FUNCTION_BLOCK TTest_LicenceCheck EXTENDS TcUnit.FB_TestSuite
VAR_INPUT
END_VAR
VAR_OUTPUT
END_VAR
VAR
END_VAR

LicenceCheck_GetsValidLicence();
LicenceCheck_GetsInValidLicence();

METHOD LicenceCheck_GetsInValidLicence
VAR_INST
    LicenceCheck : TLicenceCheck(
        LicenceIdAsString      := '{13ae39d9-bbb2-423e-8ace-d2c791a6b0ec}', // 1st digit should be 0
        LicenceName            := 'tcl_BaseLib',
        StopTwinCAT_IfNotValid := FALSE);
END_VAR
TEST(TestName := 'LicenceCheck_GetsInValidLicence');

LicenceCheck();

IF LicenceCheck.CheckComplete THEN
    AssertEquals_BOOL(
        Expected := FALSE,
        Actual   := LicenceCheck.IsValid,
        Message  := 'Licence check failed');
        
    TEST_FINISHED();
END_IF
END_METHOD

METHOD LicenceCheck_GetsValidLicence
VAR_INST
    LicenceCheck : TLicenceCheck(
        LicenceIdAsString      := '{4c256767-e6e6-4af5-bd68-9f7abad0c200}', // Tc_Ads Id
        LicenceName            := 'tcl_BaseLib',
        StopTwinCAT_IfNotValid := FALSE);
END_VAR
TEST(TestName := 'LicenceCheck_GetsValidLicence');

LicenceCheck();

IF LicenceCheck.CheckComplete THEN
    AssertEquals_BOOL(
        Expected := TRUE,
        Actual   := LicenceCheck.IsValid,
        Message  := 'Licence check failed');
        
    TEST_FINISHED();
END_IF
END_METHOD

END_FUNCTION_BLOCK

(* stored: Version 1.1.0.1, ProductVersion 3.1.4024.3
   POU TTest_LicenceCheck: Id {9134114e-323a-0056-10d4-55040573e291}, SpecialFunc None
   Method LicenceCheck_GetsInValidLicence: Id {cd10a4e4-1671-0e46-06af-1271f2891056}
   Method LicenceCheck_GetsValidLicence: Id {7393d5fc-3b1b-06b9-1054-03b3e38687bc} *)
